(* IEC 61131-3 sources: JaccoSigma/tempclass/Class/My_XAccess, 1 file *)

(* ---- My_XAccess.st ---- *)
(*!
<Class
	Name               = "My_XAccess"
	Revision           = "0.0"
	RealtimeTask       = "false"
	CyclicTask         = "false"
	BackgroundTask     = "false"
	Sigmatek           = "false"
	OSInterface        = "false"
	HighPriority       = "false"
	Automatic          = "false"
	UpdateMode         = "Prescan"
	SharedCommandTable = "true"
	Objectsize         = "(284,120)">
	<Channels>
		<Server Name="OthersHadAEvent" Visualized="true" Remotely="true" Initialize="false" WriteProtected="false" Retentive="false"/>
		<Client Name="WeHadAEvent" Required="true" Internal="false"/>
	</Channels>
	<Network Name="My_XAccess">
		<!-- List of Components in this network -->
		<Components>
			<Object
				Name       = "_base"
				Class      = "_XAccess"
				Position   = "(218,120)"
				Visualized = "true"
				Remotely   = "true">
				<Channels>
					<Server Name="Key1"/>
					<Server Name="Key2"/>
					<Server Name="Key3"/>
					<Server Name="Level"/>
					<Server Name="Server0"/>
					<Server Name="TimeOut"/>
					<Client Name="Lse"/>
				</Channels>
			</Object>
		</Components>
		<Comments>
		</Comments>
		<!-- List of Connections in this network -->
		<Connections>
			<Connection Source="this.Server0" Destination="_base.Server0" Vertices="(690,210),(518,210),"/>
			<Connection Source="this.TimeOut" Destination="_base.TimeOut" Vertices="(690,270),(518,270),"/>
			<Connection Source="this.Level" Destination="_base.Level" Vertices="(690,330),(518,330),"/>
			<Connection Source="this.Key1" Destination="_base.Key1" Vertices="(690,390),(518,390),"/>
			<Connection Source="this.Key2" Destination="_base.Key2" Vertices="(690,450),(518,450),"/>
			<Connection Source="this.Key3" Destination="_base.Key3" Vertices="(690,510),(518,510),"/>
		</Connections>
		<!-- Headerfiles -->
		<Options>
		</Options>
	</Network>
</Class>
*)
#pragma using _XAccess

My_XAccess : CLASS
: _XAccess
  //Servers:
	OthersHadAEvent 	: SvrCh_DINT;
  //Clients:
	WeHadAEvent 	: CltCh_DINT;
  //Variables:
  //Functions:

	FUNCTION VIRTUAL GLOBAL IF_WindowRun
		VAR_INPUT
			whoami 	: ^_WHOAMI;
			pic 	: ^void;
			event 	: ^_EVENT;
		END_VAR;
  //Tables:
	FUNCTION @STD
		VAR_OUTPUT
			ret_code	: CONFSTATES;
		END_VAR;
	FUNCTION GLOBAL TAB @CT_;
END_CLASS;

FUNCTION VIRTUAL GLOBAL My_XAccess::IF_WindowRun
	VAR_INPUT
		whoami 	: ^_WHOAMI;
		pic 	: ^void;
		event 	: ^_EVENT;
	END_VAR

  if(event^.ftype <> _EVENT_NONE) then
    InternTime := to_dint(Ops.tAbsolute);
    WeHadAEvent.Write(input:=1);
  elsif OthersHadAEvent <> 0 then
    InternTime := to_dint(Ops.tAbsolute);
    OthersHadAEvent := 0;
  else
    TimeOut := TO_DINT(Ram0.Read());
    if(TimeOut > 10000) then
      if((Ops.tAbsolute$DINT - InternTime) >= TimeOut) then
	      Server0 := 0;
		    CalculateLevel();
	    end_if;
    end_if;
  end_if;

END_FUNCTION //VIRTUAL GLOBAL _XAccess::IF_WindowRun
